// TIA Portal V20 export
DATA_BLOCK "CallEquipment_DB"   // DB92
{ DB_Accessible_From_OPC_UA := 'FALSE' }
// stored: AssignedProDiagFB Unit1.Em4.ProDiag, DBAccessibleFromOPCUA false, DBAccessibleFromWebserver false, InstanceOfName Unit1.Em4.CallEquipment, InstanceOfType FB, Namespace Unit1.Em4
"Unit1.Em4.CallEquipment"
   // VAR_INPUT
   //    ZoneOperationEnable { ExternalWritable := 'False'} : "LWONIK_typeSafetyZoneManualOperation";
   //    unitEnableControlInterfaces { ExternalWritable := 'False'} : "LAF_typeEnableControlInterfaces";
   //    commandExcute { ExternalWritable := 'False'} : Bool;
   // END_VAR
   // VAR_IN_OUT
   //    unitStatus : "LAF_typeUnitStatus";
   //    emFeedback : "LUC_typeEmFeedback";
   //    unitAlarmDB : "LAF_typeAlarms";
   // END_VAR
   // VAR
   //    instSequence { ExternalWritable := 'False'} : "Unit1.Em4.Sequence_1_Cutter";
   //    instCutterInitializedJob1 { ExternalWritable := 'False'} : "LAF_SelectJob";
   //    instCutterCycleJob2 { S7_SetPoint := 'True'} : "LAF_SelectJob";
   //    instCmCompensatorAxisZ { ExternalWritable := 'False'} : "LBC_AxisControl_TecPlcCn";
   //    instCmFeedingRollAxisB { ExternalWritable := 'False'} : "LBC_AxisControl_TecPlcCn";
   //    instCmElectrodeCutterAxisZ { ExternalWritable := 'False'} : "LBC_AxisControl_TecPlcCn";
   //    instCmPositionMovingAxisX { ExternalWritable := 'False'} : "LBC_Axis64Pos_TecPlcCn";
   //    instCmFeederCylinderUpDown { ExternalWritable := 'False'} : "LBC_TwoWayActuatorCn";
   //    instCmCompensatorSafetyPinIdlePosition { ExternalWritable := 'False'} : "LBC_DigitalSignalCn";
   //    instCmTabDetectSensor { ExternalWritable := 'False'} : "LBC_DigitalSignalCn";
   //    instCmTapeDetectSensor { ExternalWritable := 'False'} : "LBC_DigitalSignalCn";
   //    instCutterEpcAnalogInput { ExternalWritable := 'False'} : "LBC_AnalogInputCn";
   //    instCompensatorAxisControlInterlockSummary { ExternalWritable := 'False'} : "LER_AxisControl_InterlockSummary";
   //    instFeedingRollAxisControlInterlockSummary { ExternalWritable := 'False'} : "LER_AxisControl_InterlockSummary";
   //    instCutterAxisControlInterlockSummary { ExternalWritable := 'False'} : "LER_AxisControl_InterlockSummary";
   //    instPostionMovingAxisControlInterlockSummary { ExternalWritable := 'False'} : "LER_Axis64Pos_InterlockSummary";
   //    instServoTorqueCal_DR3 { ExternalWritable := 'False'} : "LER_ServoTorqueCal";
   //    instServoTorqueCal_DR4 { ExternalWritable := 'False'} : "LER_ServoTorqueCal";
   //    instServoTorqueCal_DR5 { ExternalWritable := 'False'} : "LER_ServoTorqueCal";
   //    instServoTorqueCal_DR6 { ExternalWritable := 'False'} : "LER_ServoTorqueCal";
   //    instLDrv701ControlCompensatorAxisZ { ExternalWritable := 'False'} : "LDrvSafe_SinaTlg701Control";
   //    instLDrv701StatusCompensatorAxisZ { ExternalWritable := 'False'} : "LDrvSafe_SinaTlg701Status";
   //    instLDrv701ControlFeedingRollAxisB { ExternalWritable := 'False'} : "LDrvSafe_SinaTlg701Control";
   //    instLDrv701StatusFeedingRollAxisB { ExternalWritable := 'False'} : "LDrvSafe_SinaTlg701Status";
   //    instLDrv701ControlElectrodeCutterAxisZ { ExternalWritable := 'False'} : "LDrvSafe_SinaTlg701Control";
   //    instLDrv701StatusElectrodeCutterAxisZ { ExternalWritable := 'False'} : "LDrvSafe_SinaTlg701Status";
   //    instLDrv701ControlPositionMovingAxisX { ExternalWritable := 'False'} : "LDrvSafe_SinaTlg701Control";
   //    instLDrv701StatusPositionMovingAxisX { ExternalWritable := 'False'} : "LDrvSafe_SinaTlg701Status";
   //    statUnitStatus { ExternalWritable := 'False'} : "LAF_typeUnitStatus";
   //    statAllBrakeTest { ExternalWritable := 'False'} : "LER_typeBrakeTestUnitCommands";
   //    instManageAlarms { ExternalWritable := 'False'} : "LAF_ManageAlarms";
   //    instEventsPFE { S7_SetPoint := 'True'} : "Unit1.Em4.EventsPFE";
   //    statPulse { ExternalWritable := 'False'} : Array[0..99] of Bool;
   //    statTonTimer { ExternalWritable := 'False'} : Array[0..99] of TON_TIME;
   //    statTofTimer { ExternalWritable := 'False'} : Array[0..99] of TOF_TIME;
   //    statEnableManualCmds { ExternalWritable := 'False'} : Bool;
   //    EndOfCycle_Complete { ExternalWritable := 'False'} : Bool;
   // END_VAR
BEGIN
END_DATA_BLOCK
